TYPE ST_GripperChannelFeedback :
STRUCT
    bBusy          : BOOL;
    udiAcceptedId  : UDINT;
    udiCompletedId : UDINT;
    udiRejectedId  : UDINT;
    udiFailedId    : UDINT;
    udErrorCode    : UDINT;
    bCloseTargetReachedWithoutGrip : BOOL; // 与udiCompletedId绑定；非Grip、非Error
END_STRUCT
END_TYPE

(* stored: Version 1.1.0.1, ProductVersion 3.1.4026.20
   DUT ST_GripperChannelFeedback: Id {f90dc80c-ec6d-40fd-a3a7-a3cf88f36ea1} *)
